Staubli VAL3: init.pgx

public program init()
  local num l_nI
  local bool l_bLoggedIn
begin
  //-----------------------------------------------------------------------
  //Header begin
  //Description of program
  //  Initialize cognex communication library.
  //  This routine must be called only once when the application is started.
  //
  //History
  //  Creation : 19-05-08 - f.Rob
  //Header end
  //-----------------------------------------------------------------------
  bDebugProgram=false
  bDebugSocket=false
  bCheckRowUpLim=true
  bGetID=false
  nLibErrorCode=0
end
